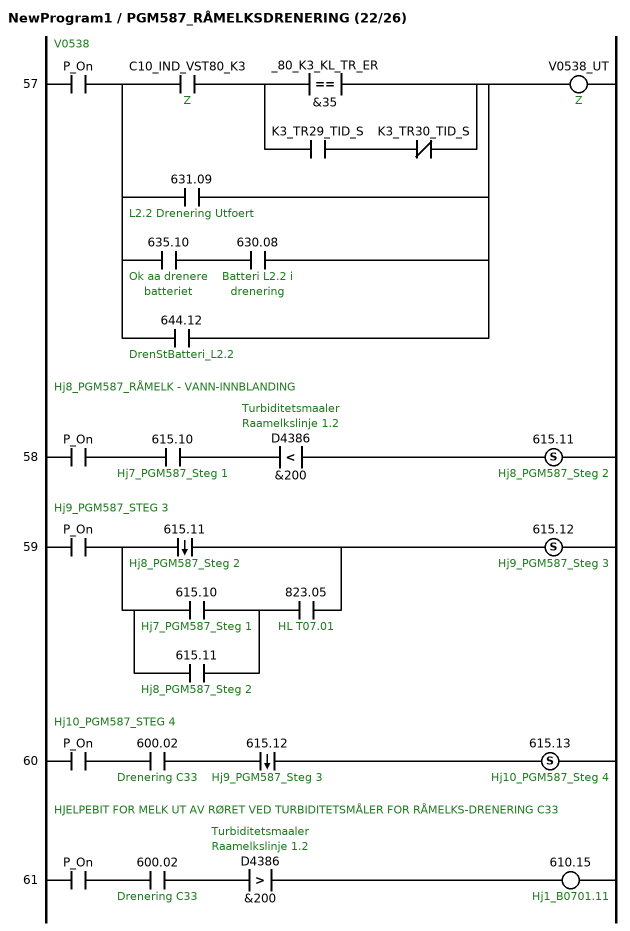
; [picture p744: NewProgram1 / PGM587_RÅMELKSDRENERING, rungs 57-61]
; rung 57: V0538
LD P_On
LD C10_IND_VST80_K3  ; Z
LD=(300) _80_K3_KL_TR_ER &35
LD K3_TR29_TID_S
ANDNOT K3_TR30_TID_S
ORLD
ANDLD
OR 631.09  ; L2.2 Drenering Utfoert
LD 635.10  ; Ok aa drenere batteriet
AND 630.08  ; Batteri L2.2 i drenering
ORLD
OR 644.12  ; DrenStBatteri_L2.2
ANDLD
OUT V0538_UT  ; Z
; rung 58: Hj8_PGM587_RÅMELK - VANN-INNBLANDING
LD P_On
AND 615.10  ; Hj7_PGM587_Steg 1
AND<(310) D4386 &200  ; Turbiditetsmaaler Raamelkslinje 1.2
SET 615.11  ; Hj8_PGM587_Steg 2
; rung 59: Hj9_PGM587_STEG 3
LD P_On
%LD 615.11  ; Hj8_PGM587_Steg 2
LD 615.10  ; Hj7_PGM587_Steg 1
OR 615.11  ; Hj8_PGM587_Steg 2
AND 823.05  ; HL T07.01
ORLD
ANDLD
SET 615.12  ; Hj9_PGM587_Steg 3
; rung 60: Hj10_PGM587_STEG 4
LD P_On
AND 600.02  ; Drenering C33
%AND 615.12  ; Hj9_PGM587_Steg 3
SET 615.13  ; Hj10_PGM587_Steg 4
; rung 61: HJELPEBIT FOR MELK UT AV RØRET VED TURBIDITETSMÅLER FOR RÅMELKS-DRENERING C33
LD P_On
AND 600.02  ; Drenering C33
AND>(320) D4386 &200  ; Turbiditetsmaaler Raamelkslinje 1.2
OUT 610.15  ; Hj1_B0701.11

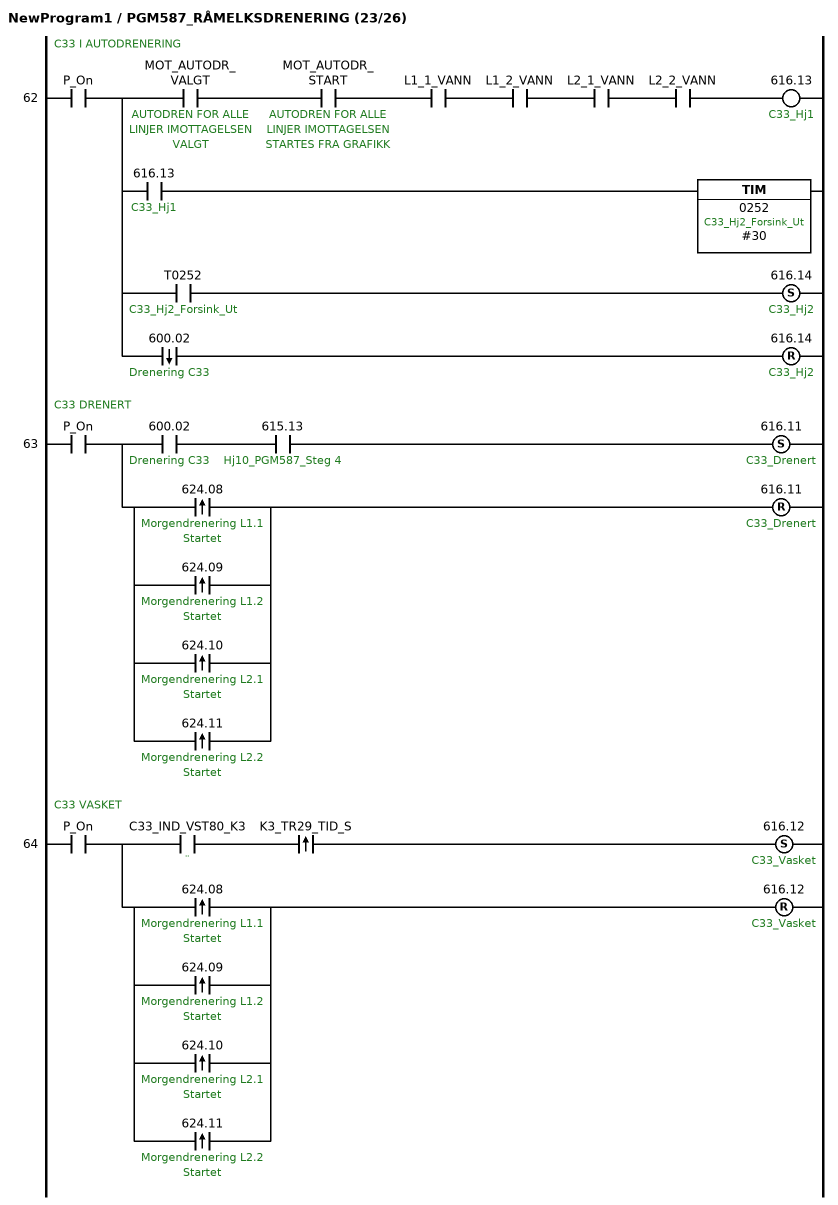
; rung 62: C33 I AUTODRENERING
LD P_On
OUT TR0
AND MOT_AUTODR_VALGT  ; AUTODREN FOR ALLE LINJER IMOTTAGELSEN VALGT
AND MOT_AUTODR_START  ; AUTODREN FOR ALLE LINJER IMOTTAGELSEN STARTES FRA GRAFIKK
AND L1_1_VANN
AND L1_2_VANN
AND L2_1_VANN
AND L2_2_VANN
OUT 616.13  ; C33_Hj1
LD TR0
AND 616.13  ; C33_Hj1
TIM 0252 #30  ; C33_Hj2_Forsink_Ut
LD TR0
AND T0252  ; C33_Hj2_Forsink_Ut
SET 616.14  ; C33_Hj2
LD TR0
%AND 600.02  ; Drenering C33
RSET 616.14  ; C33_Hj2
; rung 63: C33 DRENERT
LD P_On
OUT TR0
AND 600.02  ; Drenering C33
AND 615.13  ; Hj10_PGM587_Steg 4
SET 616.11  ; C33_Drenert
LD TR0
@LD 624.08  ; Morgendrenering L1.1 Startet
@OR 624.09  ; Morgendrenering L1.2 Startet
@OR 624.10  ; Morgendrenering L2.1 Startet
@OR 624.11  ; Morgendrenering L2.2 Startet
ANDLD
RSET 616.11  ; C33_Drenert
; rung 64: C33 VASKET
LD P_On
OUT TR0
AND C33_IND_VST80_K3  ; ¨
@AND K3_TR29_TID_S
SET 616.12  ; C33_Vasket
LD TR0
@LD 624.08  ; Morgendrenering L1.1 Startet
@OR 624.09  ; Morgendrenering L1.2 Startet
@OR 624.10  ; Morgendrenering L2.1 Startet
@OR 624.11  ; Morgendrenering L2.2 Startet
ANDLD
RSET 616.12  ; C33_Vasket

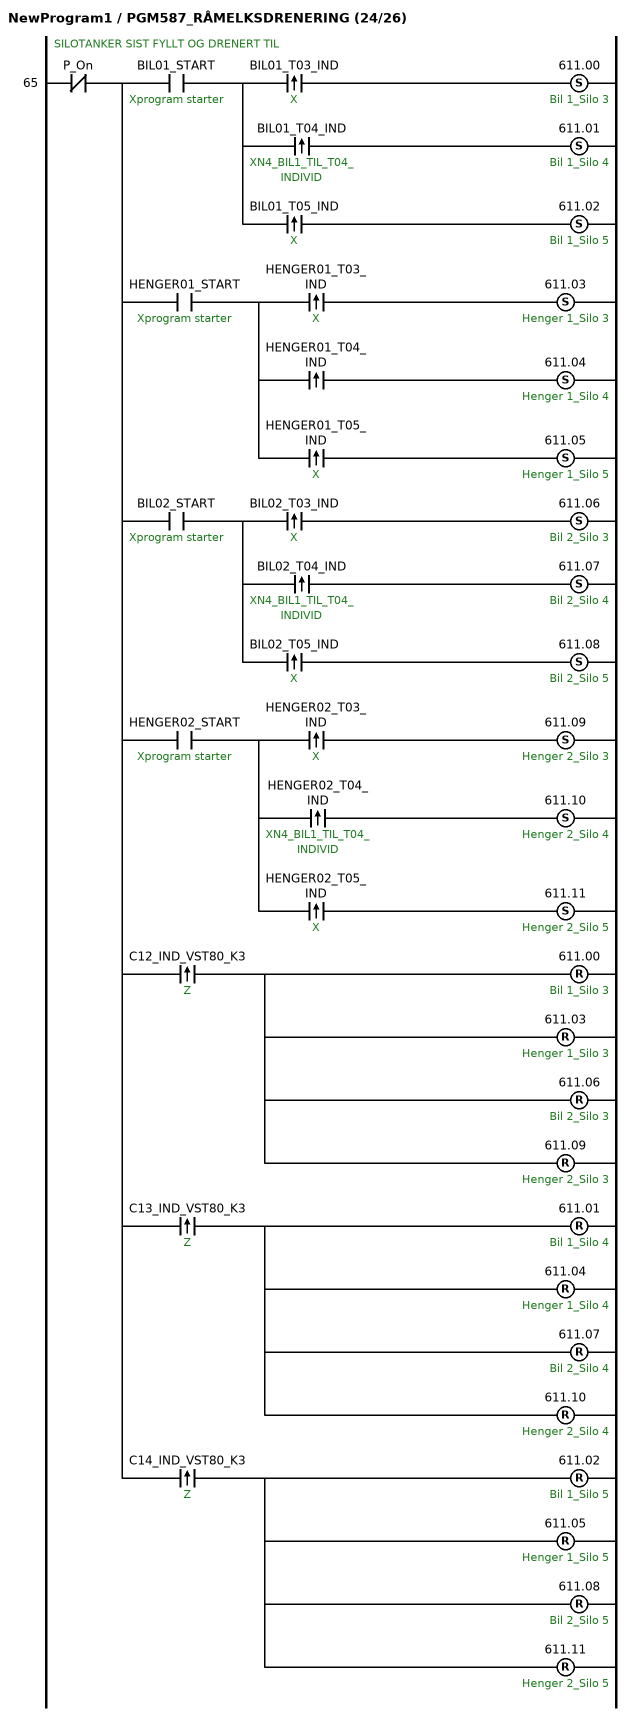
; rung 65: SILOTANKER SIST FYLLT OG DRENERT TIL
LDNOT P_On
OUT TR0
AND BIL01_START  ; Xprogram starter
OUT TR1
@AND BIL01_T03_IND  ; X
SET 611.00  ; Bil 1_Silo 3
LD TR1
@AND BIL01_T04_IND  ; XN4_BIL1_TIL_T04_INDIVID
SET 611.01  ; Bil 1_Silo 4
LD TR1
@AND BIL01_T05_IND  ; X
SET 611.02  ; Bil 1_Silo 5
LD TR0
AND HENGER01_START  ; Xprogram starter
OUT TR1
@AND HENGER01_T03_IND  ; X
SET 611.03  ; Henger 1_Silo 3
LD TR1
@AND HENGER01_T04_IND
SET 611.04  ; Henger 1_Silo 4
LD TR1
@AND HENGER01_T05_IND  ; X
SET 611.05  ; Henger 1_Silo 5
LD TR0
AND BIL02_START  ; Xprogram starter
OUT TR1
@AND BIL02_T03_IND  ; X
SET 611.06  ; Bil 2_Silo 3
LD TR1
@AND BIL02_T04_IND  ; XN4_BIL1_TIL_T04_INDIVID
SET 611.07  ; Bil 2_Silo 4
LD TR1
@AND BIL02_T05_IND  ; X
SET 611.08  ; Bil 2_Silo 5
LD TR0
AND HENGER02_START  ; Xprogram starter
OUT TR1
@AND HENGER02_T03_IND  ; X
SET 611.09  ; Henger 2_Silo 3
LD TR1
@AND HENGER02_T04_IND  ; XN4_BIL1_TIL_T04_INDIVID
SET 611.10  ; Henger 2_Silo 4
LD TR1
@AND HENGER02_T05_IND  ; X
SET 611.11  ; Henger 2_Silo 5
LD TR0
@AND C12_IND_VST80_K3  ; Z
RSET 611.00  ; Bil 1_Silo 3
RSET 611.03  ; Henger 1_Silo 3
RSET 611.06  ; Bil 2_Silo 3
RSET 611.09  ; Henger 2_Silo 3
LD TR0
@AND C13_IND_VST80_K3  ; Z
RSET 611.01  ; Bil 1_Silo 4
RSET 611.04  ; Henger 1_Silo 4
RSET 611.07  ; Bil 2_Silo 4
RSET 611.10  ; Henger 2_Silo 4
LD TR0
@AND C14_IND_VST80_K3  ; Z
RSET 611.02  ; Bil 1_Silo 5
RSET 611.05  ; Henger 1_Silo 5
RSET 611.08  ; Bil 2_Silo 5
RSET 611.11  ; Henger 2_Silo 5

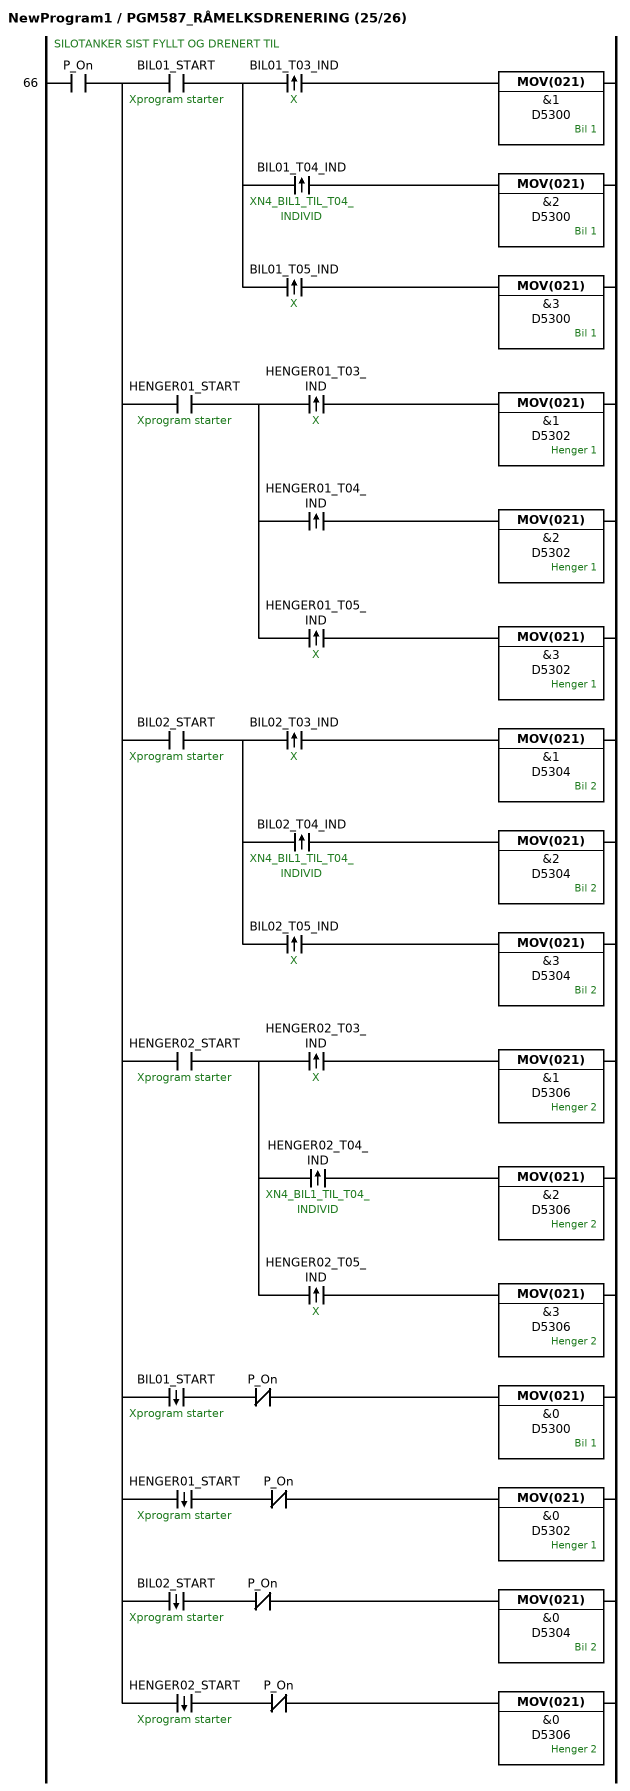
; rung 66: SILOTANKER SIST FYLLT OG DRENERT TIL
LD P_On
OUT TR0
AND BIL01_START  ; Xprogram starter
OUT TR1
@AND BIL01_T03_IND  ; X
MOV(021) &1 D5300  ; Bil 1
LD TR1
@AND BIL01_T04_IND  ; XN4_BIL1_TIL_T04_INDIVID
MOV(021) &2 D5300  ; Bil 1
LD TR1
@AND BIL01_T05_IND  ; X
MOV(021) &3 D5300  ; Bil 1
LD TR0
AND HENGER01_START  ; Xprogram starter
OUT TR1
@AND HENGER01_T03_IND  ; X
MOV(021) &1 D5302  ; Henger 1
LD TR1
@AND HENGER01_T04_IND
MOV(021) &2 D5302  ; Henger 1
LD TR1
@AND HENGER01_T05_IND  ; X
MOV(021) &3 D5302  ; Henger 1
LD TR0
AND BIL02_START  ; Xprogram starter
OUT TR1
@AND BIL02_T03_IND  ; X
MOV(021) &1 D5304  ; Bil 2
LD TR1
@AND BIL02_T04_IND  ; XN4_BIL1_TIL_T04_INDIVID
MOV(021) &2 D5304  ; Bil 2
LD TR1
@AND BIL02_T05_IND  ; X
MOV(021) &3 D5304  ; Bil 2
LD TR0
AND HENGER02_START  ; Xprogram starter
OUT TR1
@AND HENGER02_T03_IND  ; X
MOV(021) &1 D5306  ; Henger 2
LD TR1
@AND HENGER02_T04_IND  ; XN4_BIL1_TIL_T04_INDIVID
MOV(021) &2 D5306  ; Henger 2
LD TR1
@AND HENGER02_T05_IND  ; X
MOV(021) &3 D5306  ; Henger 2
LD TR0
%AND BIL01_START  ; Xprogram starter
ANDNOT P_On
MOV(021) &0 D5300  ; Bil 1
LD TR0
%AND HENGER01_START  ; Xprogram starter
ANDNOT P_On
MOV(021) &0 D5302  ; Henger 1
LD TR0
%AND BIL02_START  ; Xprogram starter
ANDNOT P_On
MOV(021) &0 D5304  ; Bil 2
LD TR0
%AND HENGER02_START  ; Xprogram starter
ANDNOT P_On
MOV(021) &0 D5306  ; Henger 2

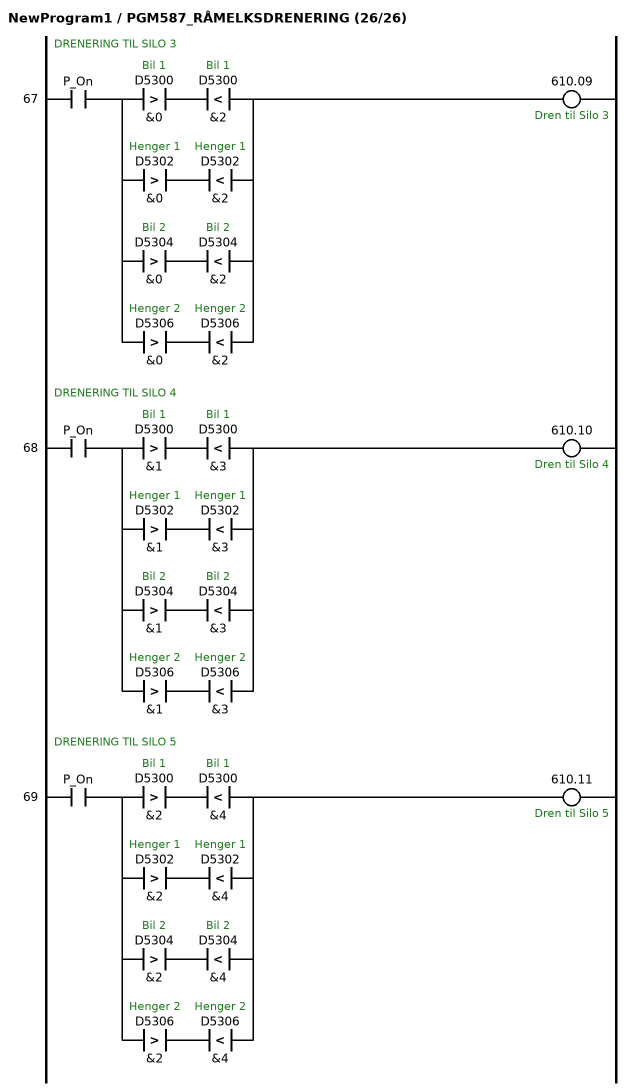
; rung 67: DRENERING TIL SILO 3
LD P_On
LD>(320) D5300 &0  ; Bil 1
AND<(310) D5300 &2  ; Bil 1
LD>(320) D5302 &0  ; Henger 1
AND<(310) D5302 &2  ; Henger 1
ORLD
LD>(320) D5304 &0  ; Bil 2
AND<(310) D5304 &2  ; Bil 2
ORLD
LD>(320) D5306 &0  ; Henger 2
AND<(310) D5306 &2  ; Henger 2
ORLD
ANDLD
OUT 610.09  ; Dren til Silo 3
; rung 68: DRENERING TIL SILO 4
LD P_On
LD>(320) D5300 &1  ; Bil 1
AND<(310) D5300 &3  ; Bil 1
LD>(320) D5302 &1  ; Henger 1
AND<(310) D5302 &3  ; Henger 1
ORLD
LD>(320) D5304 &1  ; Bil 2
AND<(310) D5304 &3  ; Bil 2
ORLD
LD>(320) D5306 &1  ; Henger 2
AND<(310) D5306 &3  ; Henger 2
ORLD
ANDLD
OUT 610.10  ; Dren til Silo 4
; rung 69: DRENERING TIL SILO 5
LD P_On
LD>(320) D5300 &2  ; Bil 1
AND<(310) D5300 &4  ; Bil 1
LD>(320) D5302 &2  ; Henger 1
AND<(310) D5302 &4  ; Henger 1
ORLD
LD>(320) D5304 &2  ; Bil 2
AND<(310) D5304 &4  ; Bil 2
ORLD
LD>(320) D5306 &2  ; Henger 2
AND<(310) D5306 &4  ; Henger 2
ORLD
ANDLD
OUT 610.11  ; Dren til Silo 5

### Section PGM588_DEPONI_T27_03

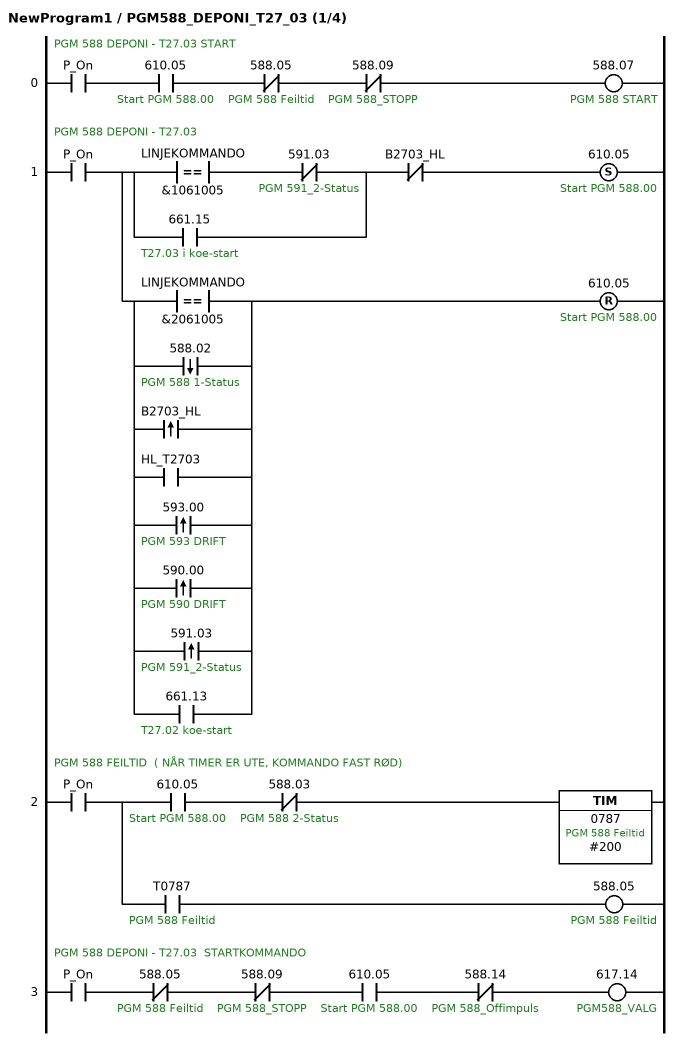
; rung 0: PGM 588 DEPONI - T27.03 START
LD P_On
AND 610.05  ; Start PGM 588.00
ANDNOT 588.05  ; PGM 588 Feiltid
ANDNOT 588.09  ; PGM 588_STOPP
OUT 588.07  ; PGM 588 START
; rung 1: PGM 588 DEPONI - T27.03
LD P_On
OUT TR0
LD=L(301) LINJEKOMMANDO &1061005
ANDNOT 591.03  ; PGM 591_2-Status
OR 661.15  ; T27.03 i koe-start
ANDLD
ANDNOT B2703_HL
SET 610.05  ; Start PGM 588.00
LD TR0
LD=L(301) LINJEKOMMANDO &2061005
%OR 588.02  ; PGM 588 1-Status
@OR B2703_HL
OR HL_T2703
@OR 593.00  ; PGM 593 DRIFT
@OR 590.00  ; PGM 590 DRIFT
@OR 591.03  ; PGM 591_2-Status
OR 661.13  ; T27.02 koe-start
ANDLD
RSET 610.05  ; Start PGM 588.00
; rung 2: PGM 588 FEILTID  ( NÅR TIMER ER UTE, KOMMANDO FAST RØD)
LD P_On
OUT TR0
AND 610.05  ; Start PGM 588.00
ANDNOT 588.03  ; PGM 588 2-Status
TIM 0787 #200  ; PGM 588 Feiltid
LD TR0
AND T0787  ; PGM 588 Feiltid
OUT 588.05  ; PGM 588 Feiltid
; rung 3: PGM 588 DEPONI - T27.03  STARTKOMMANDO
LD P_On
ANDNOT 588.05  ; PGM 588 Feiltid
ANDNOT 588.09  ; PGM 588_STOPP
AND 610.05  ; Start PGM 588.00
ANDNOT 588.14  ; PGM 588_Offimpuls
OUT 617.14  ; PGM588_VALG

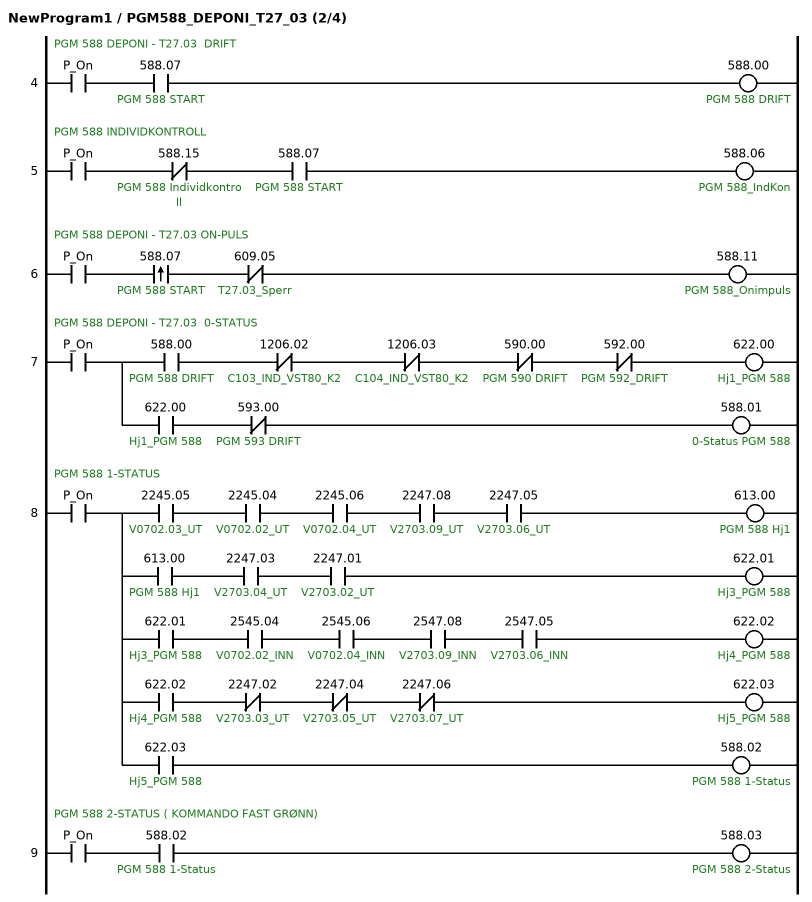
; rung 4: PGM 588 DEPONI - T27.03  DRIFT
LD P_On
AND 588.07  ; PGM 588 START
OUT 588.00  ; PGM 588 DRIFT
; rung 5: PGM 588 INDIVIDKONTROLL
LD P_On
ANDNOT 588.15  ; PGM 588 Individkontroll
AND 588.07  ; PGM 588 START
OUT 588.06  ; PGM 588_IndKon
; rung 6: PGM 588 DEPONI - T27.03 ON-PULS
LD P_On
@AND 588.07  ; PGM 588 START
ANDNOT 609.05  ; T27.03_Sperr
OUT 588.11  ; PGM 588_Onimpuls
; rung 7: PGM 588 DEPONI - T27.03  0-STATUS
LD P_On
OUT TR0
AND 588.00  ; PGM 588 DRIFT
ANDNOT 1206.02  ; C103_IND_VST80_K2
ANDNOT 1206.03  ; C104_IND_VST80_K2
ANDNOT 590.00  ; PGM 590 DRIFT
ANDNOT 592.00  ; PGM 592_DRIFT
OUT 622.00  ; Hj1_PGM 588
LD TR0
AND 622.00  ; Hj1_PGM 588
ANDNOT 593.00  ; PGM 593 DRIFT
OUT 588.01  ; 0-Status PGM 588
; rung 8: PGM 588 1-STATUS
LD P_On
OUT TR0
AND 2245.05  ; V0702.03_UT
AND 2245.04  ; V0702.02_UT
AND 2245.06  ; V0702.04_UT
AND 2247.08  ; V2703.09_UT
AND 2247.05  ; V2703.06_UT
OUT 613.00  ; PGM 588 Hj1
LD TR0
AND 613.00  ; PGM 588 Hj1
AND 2247.03  ; V2703.04_UT
AND 2247.01  ; V2703.02_UT
OUT 622.01  ; Hj3_PGM 588
LD TR0
AND 622.01  ; Hj3_PGM 588
AND 2545.04  ; V0702.02_INN
AND 2545.06  ; V0702.04_INN
AND 2547.08  ; V2703.09_INN
AND 2547.05  ; V2703.06_INN
OUT 622.02  ; Hj4_PGM 588
LD TR0
AND 622.02  ; Hj4_PGM 588
ANDNOT 2247.02  ; V2703.03_UT
ANDNOT 2247.04  ; V2703.05_UT
ANDNOT 2247.06  ; V2703.07_UT
OUT 622.03  ; Hj5_PGM 588
LD TR0
AND 622.03  ; Hj5_PGM 588
OUT 588.02  ; PGM 588 1-Status
; rung 9: PGM 588 2-STATUS ( KOMMANDO FAST GRØNN)
LD P_On
AND 588.02  ; PGM 588 1-Status
OUT 588.03  ; PGM 588 2-Status

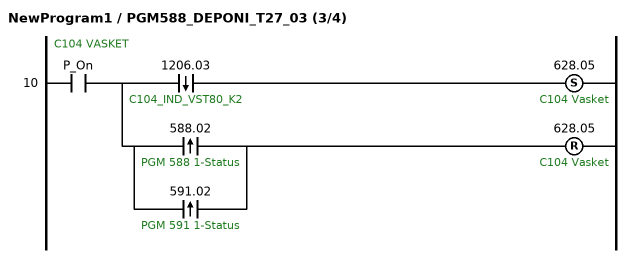
; rung 10: C104 VASKET
LD P_On
OUT TR0
%AND 1206.03  ; C104_IND_VST80_K2
SET 628.05  ; C104 Vasket
LD TR0
@LD 588.02  ; PGM 588 1-Status
@OR 591.02  ; PGM 591 1-Status
ANDLD
RSET 628.05  ; C104 Vasket

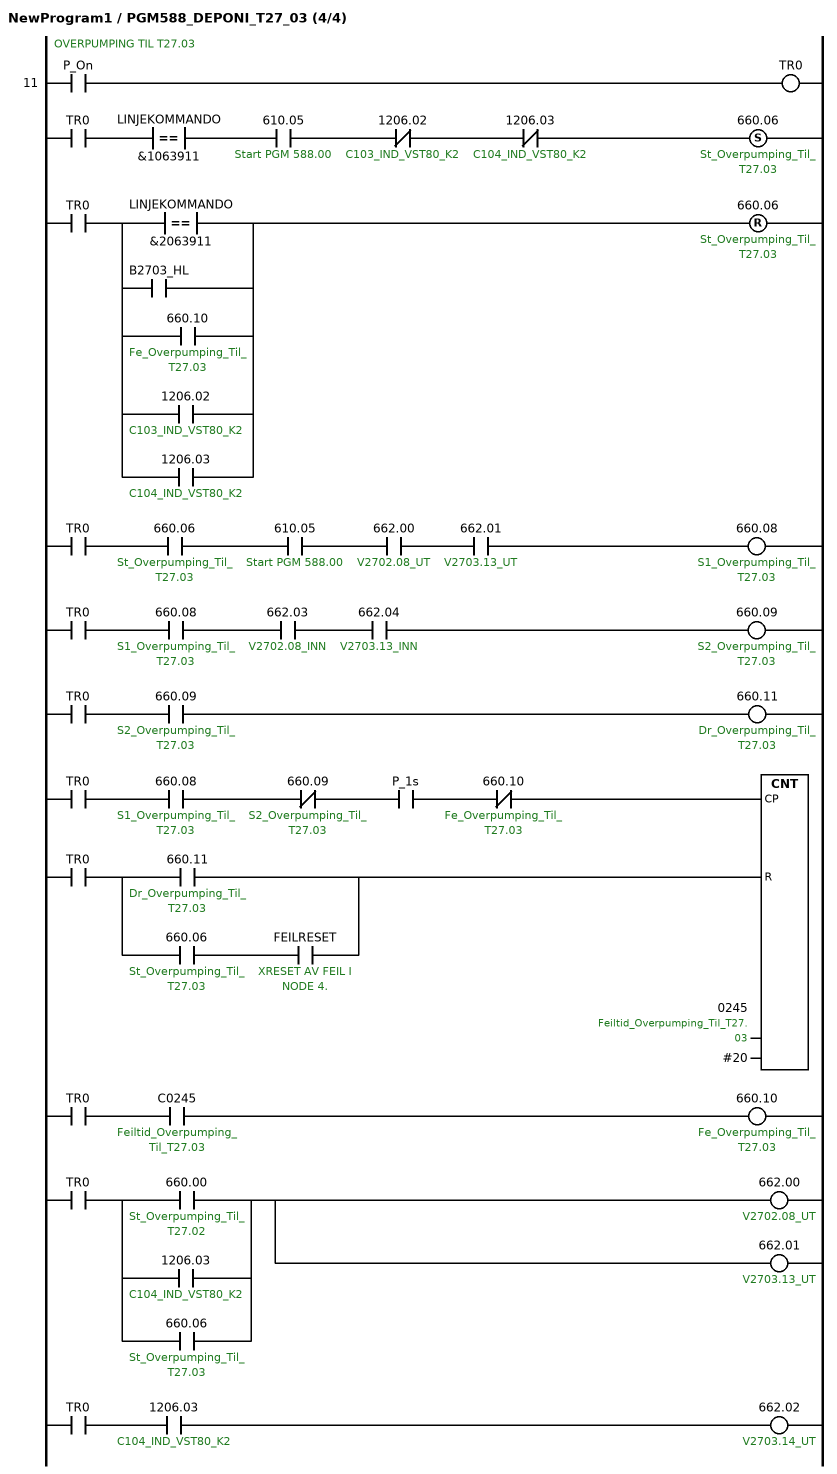
; rung 11: OVERPUMPING TIL T27.03
LD P_On
OUT TR0
AND=L(301) LINJEKOMMANDO &1063911
AND 610.05  ; Start PGM 588.00
ANDNOT 1206.02  ; C103_IND_VST80_K2
ANDNOT 1206.03  ; C104_IND_VST80_K2
SET 660.06  ; St_Overpumping_Til_T27.03
LD TR0
LD=L(301) LINJEKOMMANDO &2063911
OR B2703_HL
OR 660.10  ; Fe_Overpumping_Til_T27.03
OR 1206.02  ; C103_IND_VST80_K2
OR 1206.03  ; C104_IND_VST80_K2
ANDLD
RSET 660.06  ; St_Overpumping_Til_T27.03
LD TR0
AND 660.06  ; St_Overpumping_Til_T27.03
AND 610.05  ; Start PGM 588.00
AND 662.00  ; V2702.08_UT
AND 662.01  ; V2703.13_UT
OUT 660.08  ; S1_Overpumping_Til_T27.03
LD TR0
AND 660.08  ; S1_Overpumping_Til_T27.03
AND 662.03  ; V2702.08_INN
AND 662.04  ; V2703.13_INN
OUT 660.09  ; S2_Overpumping_Til_T27.03
LD TR0
AND 660.09  ; S2_Overpumping_Til_T27.03
OUT 660.11  ; Dr_Overpumping_Til_T27.03
LD TR0
AND 660.08  ; S1_Overpumping_Til_T27.03
ANDNOT 660.09  ; S2_Overpumping_Til_T27.03
AND P_1s
ANDNOT 660.10  ; Fe_Overpumping_Til_T27.03
LD TR0
LD 660.11  ; Dr_Overpumping_Til_T27.03
LD 660.06  ; St_Overpumping_Til_T27.03
AND FEILRESET  ; XRESET AV FEIL I NODE 4.
ORLD
ANDLD
CNT 0245 #20  ; Feiltid_Overpumping_Til_T27.03
LD TR0
AND C0245  ; Feiltid_Overpumping_Til_T27.03
OUT 660.10  ; Fe_Overpumping_Til_T27.03
LD TR0
LD 660.00  ; St_Overpumping_Til_T27.02
OR 1206.03  ; C104_IND_VST80_K2
OR 660.06  ; St_Overpumping_Til_T27.03
ANDLD
OUT 662.00  ; V2702.08_UT
OUT 662.01  ; V2703.13_UT
LD TR0
AND 1206.03  ; C104_IND_VST80_K2
OUT 662.02  ; V2703.14_UT

### Section PGM589_T27_02

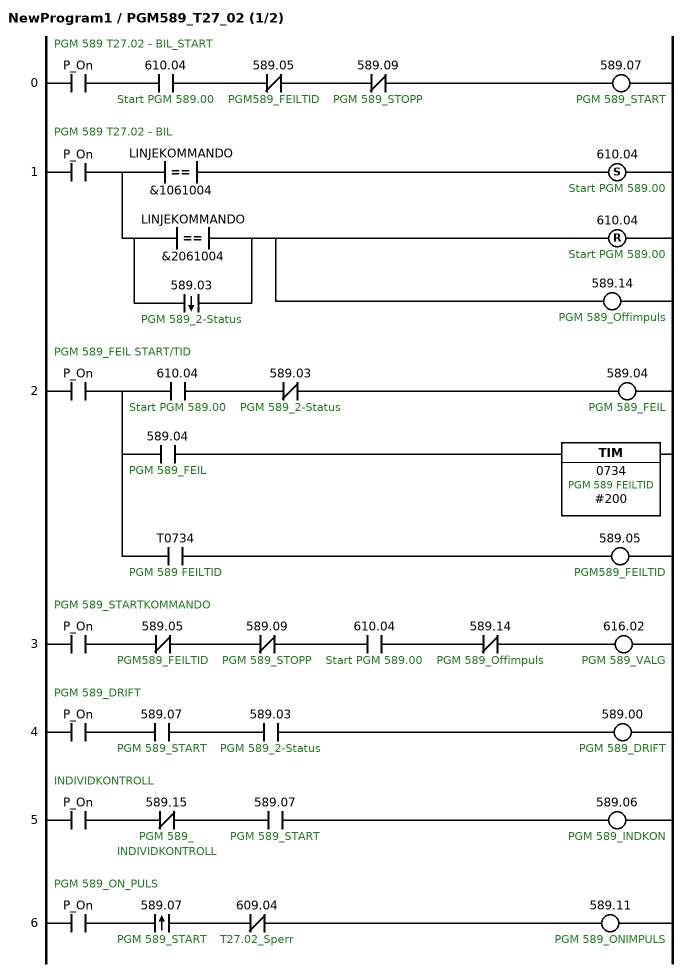
; rung 0: PGM 589 T27.02 - BIL_START
LD P_On
AND 610.04  ; Start PGM 589.00
ANDNOT 589.05  ; PGM589_FEILTID
ANDNOT 589.09  ; PGM 589_STOPP
OUT 589.07  ; PGM 589_START
; rung 1: PGM 589 T27.02 - BIL
LD P_On
OUT TR0
AND=L(301) LINJEKOMMANDO &1061004
SET 610.04  ; Start PGM 589.00
LD TR0
LD=L(301) LINJEKOMMANDO &2061004
%OR 589.03  ; PGM 589_2-Status
ANDLD
RSET 610.04  ; Start PGM 589.00
OUT 589.14  ; PGM 589_Offimpuls
; rung 2: PGM 589_FEIL START/TID
LD P_On
OUT TR0
AND 610.04  ; Start PGM 589.00
ANDNOT 589.03  ; PGM 589_2-Status
OUT 589.04  ; PGM 589_FEIL
LD TR0
AND 589.04  ; PGM 589_FEIL
TIM 0734 #200  ; PGM 589 FEILTID
LD TR0
AND T0734  ; PGM 589 FEILTID
OUT 589.05  ; PGM589_FEILTID
; rung 3: PGM 589_STARTKOMMANDO
LD P_On
ANDNOT 589.05  ; PGM589_FEILTID
ANDNOT 589.09  ; PGM 589_STOPP
AND 610.04  ; Start PGM 589.00
ANDNOT 589.14  ; PGM 589_Offimpuls
OUT 616.02  ; PGM 589_VALG
; rung 4: PGM 589_DRIFT
LD P_On
AND 589.07  ; PGM 589_START
AND 589.03  ; PGM 589_2-Status
OUT 589.00  ; PGM 589_DRIFT
; rung 5: INDIVIDKONTROLL
LD P_On
ANDNOT 589.15  ; PGM 589_INDIVIDKONTROLL
AND 589.07  ; PGM 589_START
OUT 589.06  ; PGM 589_INDKON
; rung 6: PGM 589_ON_PULS
LD P_On
@AND 589.07  ; PGM 589_START
ANDNOT 609.04  ; T27.02_Sperr
OUT 589.11  ; PGM 589_ONIMPULS

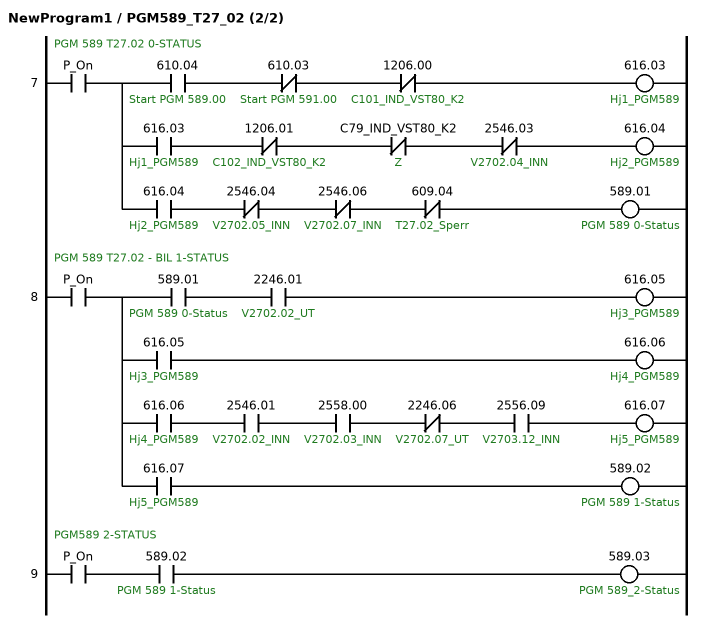
; rung 7: PGM 589 T27.02 0-STATUS
LD P_On
OUT TR0
AND 610.04  ; Start PGM 589.00
ANDNOT 610.03  ; Start PGM 591.00
ANDNOT 1206.00  ; C101_IND_VST80_K2
OUT 616.03  ; Hj1_PGM589
LD TR0
AND 616.03  ; Hj1_PGM589
ANDNOT 1206.01  ; C102_IND_VST80_K2
ANDNOT C79_IND_VST80_K2  ; Z
ANDNOT 2546.03  ; V2702.04_INN
OUT 616.04  ; Hj2_PGM589
LD TR0
AND 616.04  ; Hj2_PGM589
ANDNOT 2546.04  ; V2702.05_INN
ANDNOT 2546.06  ; V2702.07_INN
ANDNOT 609.04  ; T27.02_Sperr
OUT 589.01  ; PGM 589 0-Status
; rung 8: PGM 589 T27.02 - BIL 1-STATUS
LD P_On
OUT TR0
AND 589.01  ; PGM 589 0-Status
AND 2246.01  ; V2702.02_UT
OUT 616.05  ; Hj3_PGM589
LD TR0
AND 616.05  ; Hj3_PGM589
OUT 616.06  ; Hj4_PGM589
LD TR0
AND 616.06  ; Hj4_PGM589
AND 2546.01  ; V2702.02_INN
AND 2558.00  ; V2702.03_INN
ANDNOT 2246.06  ; V2702.07_UT
AND 2556.09  ; V2703.12_INN
OUT 616.07  ; Hj5_PGM589
LD TR0
AND 616.07  ; Hj5_PGM589
OUT 589.02  ; PGM 589 1-Status
; rung 9: PGM589 2-STATUS
LD P_On
AND 589.02  ; PGM 589 1-Status
OUT 589.03  ; PGM 589_2-Status

### Section PGM590_T27_03_BIL

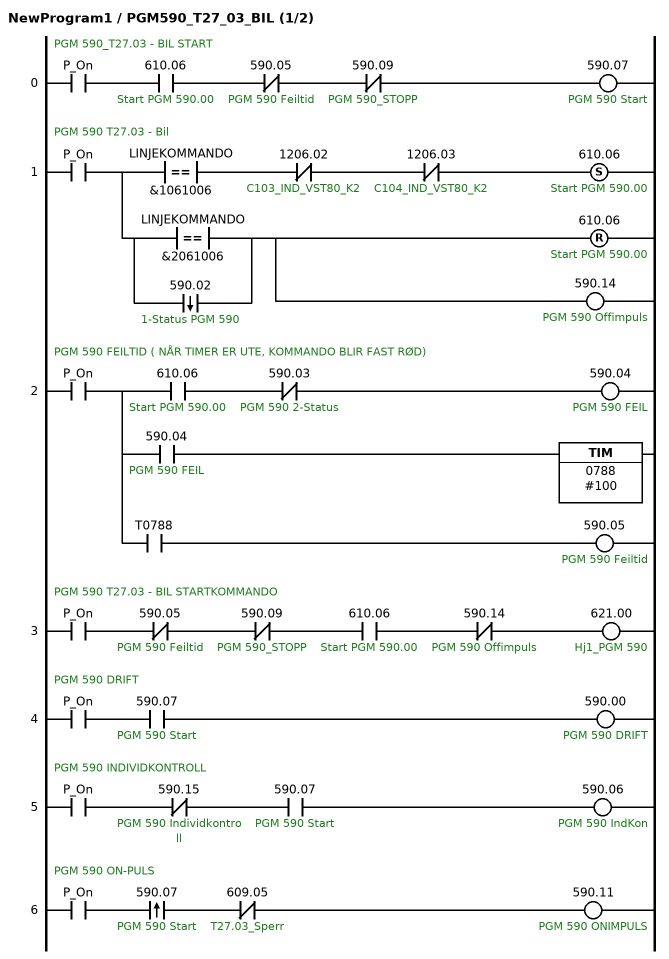
; rung 0: PGM 590_T27.03 - BIL START
LD P_On
AND 610.06  ; Start PGM 590.00
ANDNOT 590.05  ; PGM 590 Feiltid
ANDNOT 590.09  ; PGM 590_STOPP
OUT 590.07  ; PGM 590 Start
; rung 1: PGM 590 T27.03 - Bil
LD P_On
OUT TR0
AND=L(301) LINJEKOMMANDO &1061006
ANDNOT 1206.02  ; C103_IND_VST80_K2
ANDNOT 1206.03  ; C104_IND_VST80_K2
SET 610.06  ; Start PGM 590.00
LD TR0
LD=L(301) LINJEKOMMANDO &2061006
%OR 590.02  ; 1-Status PGM 590
ANDLD
RSET 610.06  ; Start PGM 590.00
OUT 590.14  ; PGM 590 Offimpuls
; rung 2: PGM 590 FEILTID ( NÅR TIMER ER UTE, KOMMANDO BLIR FAST RØD)
LD P_On
OUT TR0
AND 610.06  ; Start PGM 590.00
ANDNOT 590.03  ; PGM 590 2-Status
OUT 590.04  ; PGM 590 FEIL
LD TR0
AND 590.04  ; PGM 590 FEIL
TIM 0788 #100
LD TR0
AND T0788
OUT 590.05  ; PGM 590 Feiltid
; rung 3: PGM 590 T27.03 - BIL STARTKOMMANDO
LD P_On
ANDNOT 590.05  ; PGM 590 Feiltid
ANDNOT 590.09  ; PGM 590_STOPP
AND 610.06  ; Start PGM 590.00
ANDNOT 590.14  ; PGM 590 Offimpuls
OUT 621.00  ; Hj1_PGM 590
; rung 4: PGM 590 DRIFT
LD P_On
AND 590.07  ; PGM 590 Start
OUT 590.00  ; PGM 590 DRIFT
; rung 5: PGM 590 INDIVIDKONTROLL
LD P_On
ANDNOT 590.15  ; PGM 590 Individkontroll
AND 590.07  ; PGM 590 Start
OUT 590.06  ; PGM 590 IndKon
; rung 6: PGM 590 ON-PULS
LD P_On
@AND 590.07  ; PGM 590 Start
ANDNOT 609.05  ; T27.03_Sperr
OUT 590.11  ; PGM 590 ONIMPULS

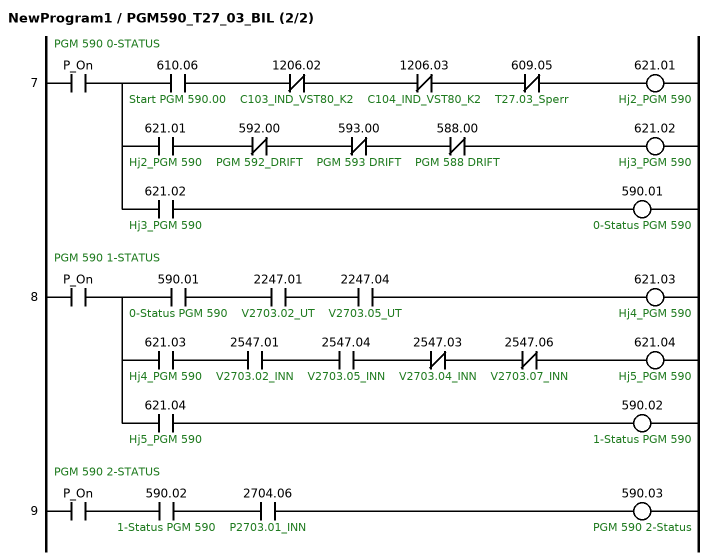
; rung 7: PGM 590 0-STATUS
LD P_On
OUT TR0
AND 610.06  ; Start PGM 590.00
ANDNOT 1206.02  ; C103_IND_VST80_K2
ANDNOT 1206.03  ; C104_IND_VST80_K2
ANDNOT 609.05  ; T27.03_Sperr
OUT 621.01  ; Hj2_PGM 590
LD TR0
AND 621.01  ; Hj2_PGM 590
ANDNOT 592.00  ; PGM 592_DRIFT
ANDNOT 593.00  ; PGM 593 DRIFT
ANDNOT 588.00  ; PGM 588 DRIFT
OUT 621.02  ; Hj3_PGM 590
LD TR0
AND 621.02  ; Hj3_PGM 590
OUT 590.01  ; 0-Status PGM 590
; rung 8: PGM 590 1-STATUS
LD P_On
OUT TR0
AND 590.01  ; 0-Status PGM 590
AND 2247.01  ; V2703.02_UT
AND 2247.04  ; V2703.05_UT
OUT 621.03  ; Hj4_PGM 590
LD TR0
AND 621.03  ; Hj4_PGM 590
AND 2547.01  ; V2703.02_INN
AND 2547.04  ; V2703.05_INN
ANDNOT 2547.03  ; V2703.04_INN
ANDNOT 2547.06  ; V2703.07_INN
OUT 621.04  ; Hj5_PGM 590
LD TR0
AND 621.04  ; Hj5_PGM 590
OUT 590.02  ; 1-Status PGM 590
; rung 9: PGM 590 2-STATUS
LD P_On
AND 590.02  ; 1-Status PGM 590
AND 2704.06  ; P2703.01_INN
OUT 590.03  ; PGM 590 2-Status

### Section PGM591_T27_02

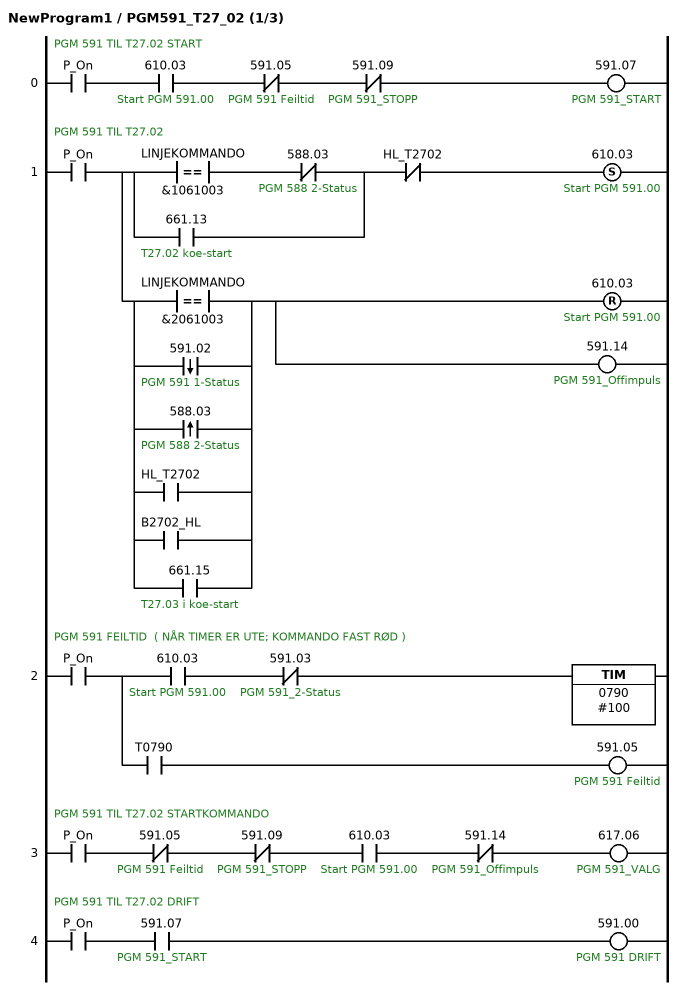
; rung 0: PGM 591 TIL T27.02 START
LD P_On
AND 610.03  ; Start PGM 591.00
ANDNOT 591.05  ; PGM 591 Feiltid
ANDNOT 591.09  ; PGM 591_STOPP
OUT 591.07  ; PGM 591_START
; rung 1: PGM 591 TIL T27.02
LD P_On
OUT TR0
LD=L(301) LINJEKOMMANDO &1061003
ANDNOT 588.03  ; PGM 588 2-Status
OR 661.13  ; T27.02 koe-start
ANDLD
ANDNOT HL_T2702
SET 610.03  ; Start PGM 591.00
LD TR0
LD=L(301) LINJEKOMMANDO &2061003
%OR 591.02  ; PGM 591 1-Status
@OR 588.03  ; PGM 588 2-Status
OR HL_T2702
OR B2702_HL
OR 661.15  ; T27.03 i koe-start
ANDLD
RSET 610.03  ; Start PGM 591.00
OUT 591.14  ; PGM 591_Offimpuls
; rung 2: PGM 591 FEILTID  ( NÅR TIMER ER UTE; KOMMANDO FAST RØD )
LD P_On
OUT TR0
AND 610.03  ; Start PGM 591.00
ANDNOT 591.03  ; PGM 591_2-Status
TIM 0790 #100
LD TR0
AND T0790
OUT 591.05  ; PGM 591 Feiltid
; rung 3: PGM 591 TIL T27.02 STARTKOMMANDO
LD P_On
ANDNOT 591.05  ; PGM 591 Feiltid
ANDNOT 591.09  ; PGM 591_STOPP
AND 610.03  ; Start PGM 591.00
ANDNOT 591.14  ; PGM 591_Offimpuls
OUT 617.06  ; PGM 591_VALG
; rung 4: PGM 591 TIL T27.02 DRIFT
LD P_On
AND 591.07  ; PGM 591_START
OUT 591.00  ; PGM 591 DRIFT

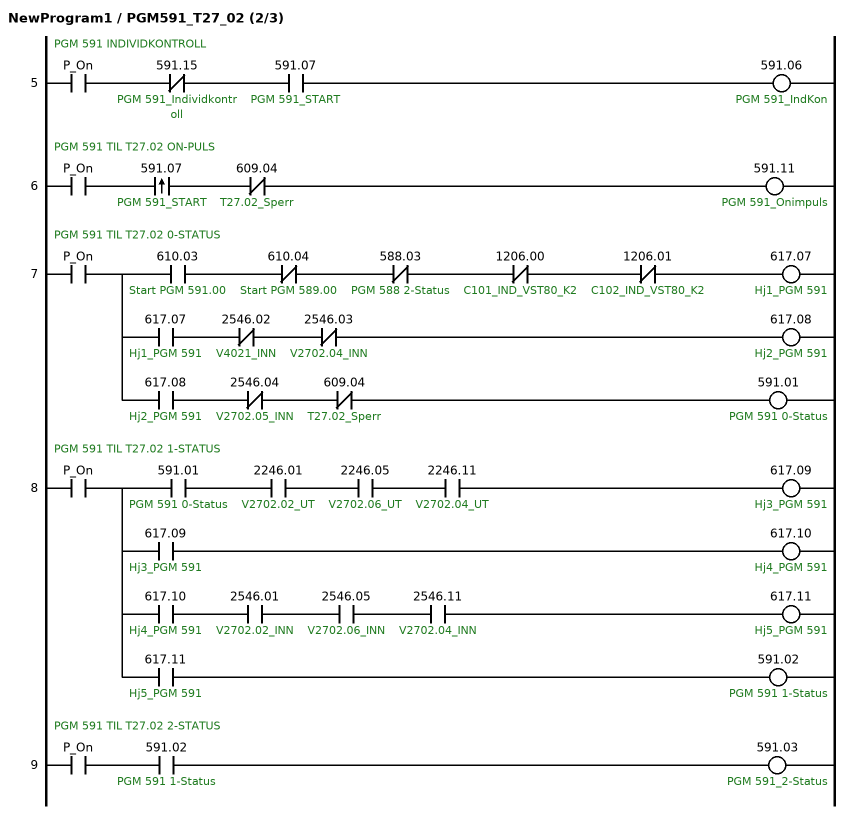
; rung 5: PGM 591 INDIVIDKONTROLL
LD P_On
ANDNOT 591.15  ; PGM 591_Individkontroll
AND 591.07  ; PGM 591_START
OUT 591.06  ; PGM 591_IndKon
; rung 6: PGM 591 TIL T27.02 ON-PULS
LD P_On
@AND 591.07  ; PGM 591_START
ANDNOT 609.04  ; T27.02_Sperr
OUT 591.11  ; PGM 591_Onimpuls
; rung 7: PGM 591 TIL T27.02 0-STATUS
LD P_On
OUT TR0
AND 610.03  ; Start PGM 591.00
ANDNOT 610.04  ; Start PGM 589.00
ANDNOT 588.03  ; PGM 588 2-Status
ANDNOT 1206.00  ; C101_IND_VST80_K2
ANDNOT 1206.01  ; C102_IND_VST80_K2
OUT 617.07  ; Hj1_PGM 591
LD TR0
AND 617.07  ; Hj1_PGM 591
ANDNOT 2546.02  ; V4021_INN
ANDNOT 2546.03  ; V2702.04_INN
OUT 617.08  ; Hj2_PGM 591
LD TR0
AND 617.08  ; Hj2_PGM 591
ANDNOT 2546.04  ; V2702.05_INN
ANDNOT 609.04  ; T27.02_Sperr
OUT 591.01  ; PGM 591 0-Status
; rung 8: PGM 591 TIL T27.02 1-STATUS
LD P_On
OUT TR0
AND 591.01  ; PGM 591 0-Status
AND 2246.01  ; V2702.02_UT
AND 2246.05  ; V2702.06_UT
AND 2246.11  ; V2702.04_UT
OUT 617.09  ; Hj3_PGM 591
LD TR0
AND 617.09  ; Hj3_PGM 591
OUT 617.10  ; Hj4_PGM 591
LD TR0
AND 617.10  ; Hj4_PGM 591
AND 2546.01  ; V2702.02_INN
AND 2546.05  ; V2702.06_INN
AND 2546.11  ; V2702.04_INN
OUT 617.11  ; Hj5_PGM 591
LD TR0
AND 617.11  ; Hj5_PGM 591
OUT 591.02  ; PGM 591 1-Status
; rung 9: PGM 591 TIL T27.02 2-STATUS
LD P_On
AND 591.02  ; PGM 591 1-Status
OUT 591.03  ; PGM 591_2-Status

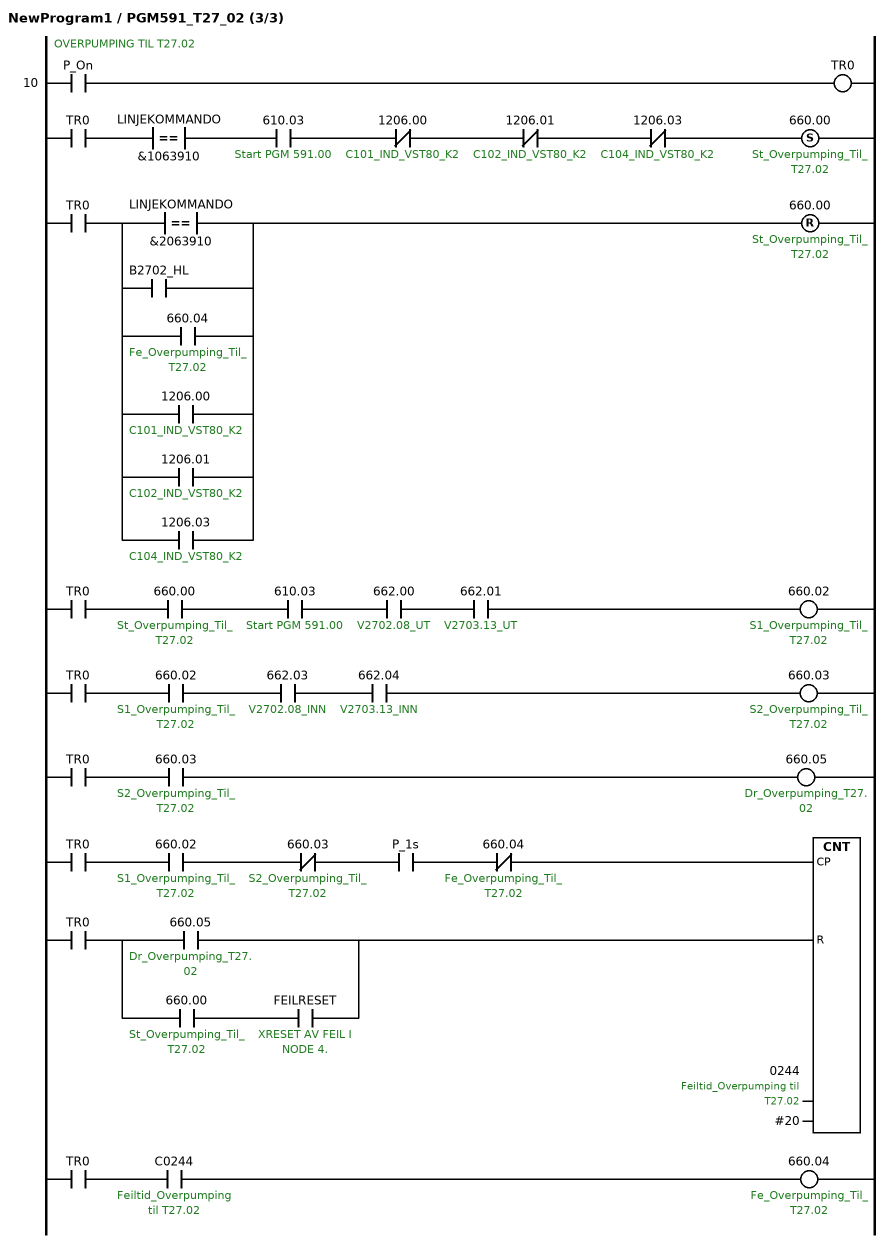
; rung 10: OVERPUMPING TIL T27.02
LD P_On
OUT TR0
AND=L(301) LINJEKOMMANDO &1063910
AND 610.03  ; Start PGM 591.00
ANDNOT 1206.00  ; C101_IND_VST80_K2
ANDNOT 1206.01  ; C102_IND_VST80_K2
ANDNOT 1206.03  ; C104_IND_VST80_K2
SET 660.00  ; St_Overpumping_Til_T27.02
LD TR0
LD=L(301) LINJEKOMMANDO &2063910
OR B2702_HL
OR 660.04  ; Fe_Overpumping_Til_T27.02
OR 1206.00  ; C101_IND_VST80_K2
OR 1206.01  ; C102_IND_VST80_K2
OR 1206.03  ; C104_IND_VST80_K2
ANDLD
RSET 660.00  ; St_Overpumping_Til_T27.02
LD TR0
AND 660.00  ; St_Overpumping_Til_T27.02
AND 610.03  ; Start PGM 591.00
AND 662.00  ; V2702.08_UT
AND 662.01  ; V2703.13_UT
OUT 660.02  ; S1_Overpumping_Til_T27.02
LD TR0
AND 660.02  ; S1_Overpumping_Til_T27.02
AND 662.03  ; V2702.08_INN
AND 662.04  ; V2703.13_INN
OUT 660.03  ; S2_Overpumping_Til_T27.02
LD TR0
AND 660.03  ; S2_Overpumping_Til_T27.02
OUT 660.05  ; Dr_Overpumping_T27.02
LD TR0
AND 660.02  ; S1_Overpumping_Til_T27.02
ANDNOT 660.03  ; S2_Overpumping_Til_T27.02
AND P_1s
ANDNOT 660.04  ; Fe_Overpumping_Til_T27.02
LD TR0
LD 660.05  ; Dr_Overpumping_T27.02
LD 660.00  ; St_Overpumping_Til_T27.02
AND FEILRESET  ; XRESET AV FEIL I NODE 4.
ORLD
ANDLD
CNT 0244 #20  ; Feiltid_Overpumping til T27.02
LD TR0
AND C0244  ; Feiltid_Overpumping til T27.02
OUT 660.04  ; Fe_Overpumping_Til_T27.02

### Section PGM592_DRENERING_T27_03

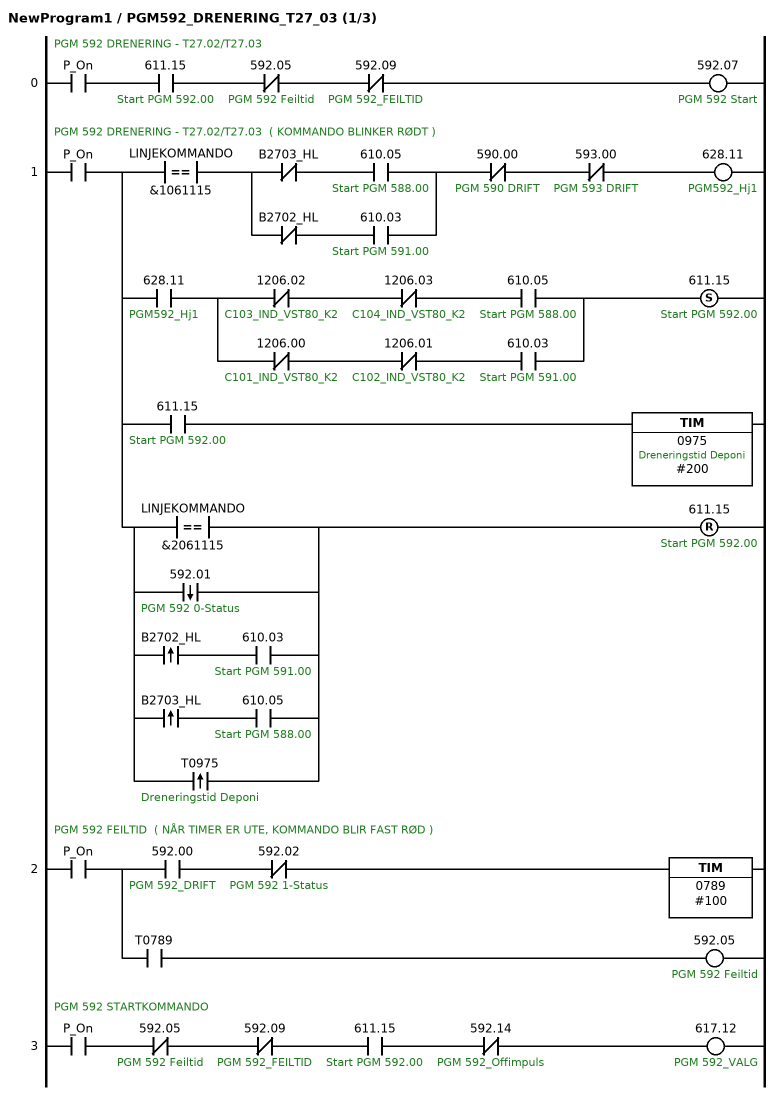
; rung 0: PGM 592 DRENERING - T27.02/T27.03
LD P_On
AND 611.15  ; Start PGM 592.00
ANDNOT 592.05  ; PGM 592 Feiltid
ANDNOT 592.09  ; PGM 592_FEILTID
OUT 592.07  ; PGM 592 Start
; rung 1: PGM 592 DRENERING - T27.02/T27.03  ( KOMMANDO BLINKER RØDT )
LD P_On
OUT TR0
AND=L(301) LINJEKOMMANDO &1061115
LDNOT B2703_HL
AND 610.05  ; Start PGM 588.00
LDNOT B2702_HL
AND 610.03  ; Start PGM 591.00
ORLD
ANDLD
ANDNOT 590.00  ; PGM 590 DRIFT
ANDNOT 593.00  ; PGM 593 DRIFT
OUT 628.11  ; PGM592_Hj1
LD TR0
AND 628.11  ; PGM592_Hj1
LDNOT 1206.02  ; C103_IND_VST80_K2
ANDNOT 1206.03  ; C104_IND_VST80_K2
AND 610.05  ; Start PGM 588.00
LDNOT 1206.00  ; C101_IND_VST80_K2
ANDNOT 1206.01  ; C102_IND_VST80_K2
AND 610.03  ; Start PGM 591.00
ORLD
ANDLD
SET 611.15  ; Start PGM 592.00
LD TR0
AND 611.15  ; Start PGM 592.00
TIM 0975 #200  ; Dreneringstid Deponi
LD TR0
LD=L(301) LINJEKOMMANDO &2061115
%OR 592.01  ; PGM 592 0-Status
@LD B2702_HL
AND 610.03  ; Start PGM 591.00
ORLD
@LD B2703_HL
AND 610.05  ; Start PGM 588.00
ORLD
@OR T0975  ; Dreneringstid Deponi
ANDLD
RSET 611.15  ; Start PGM 592.00
; rung 2: PGM 592 FEILTID  ( NÅR TIMER ER UTE, KOMMANDO BLIR FAST RØD )
LD P_On
OUT TR0
AND 592.00  ; PGM 592_DRIFT
ANDNOT 592.02  ; PGM 592 1-Status
TIM 0789 #100
LD TR0
AND T0789
OUT 592.05  ; PGM 592 Feiltid
; rung 3: PGM 592 STARTKOMMANDO
LD P_On
ANDNOT 592.05  ; PGM 592 Feiltid
ANDNOT 592.09  ; PGM 592_FEILTID
AND 611.15  ; Start PGM 592.00
ANDNOT 592.14  ; PGM 592_Offimpuls
OUT 617.12  ; PGM 592_VALG

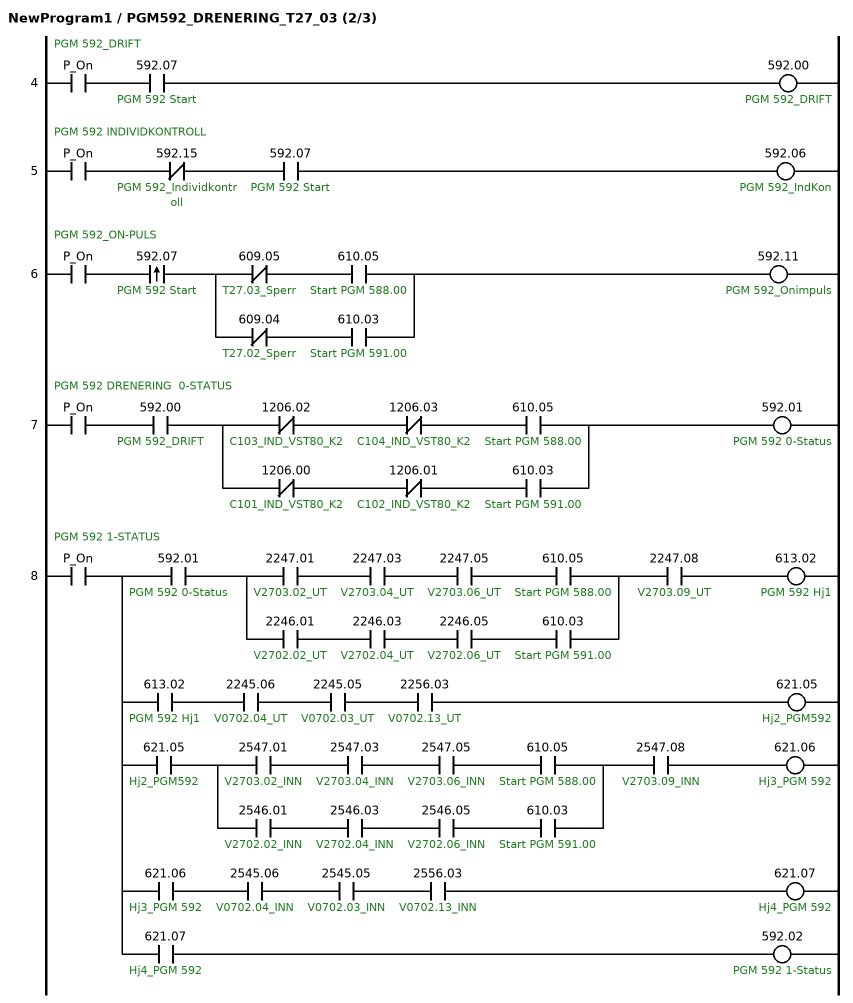
; rung 4: PGM 592_DRIFT
LD P_On
AND 592.07  ; PGM 592 Start
OUT 592.00  ; PGM 592_DRIFT
; rung 5: PGM 592 INDIVIDKONTROLL
LD P_On
ANDNOT 592.15  ; PGM 592_Individkontroll
AND 592.07  ; PGM 592 Start
OUT 592.06  ; PGM 592_IndKon
; rung 6: PGM 592_ON-PULS
LD P_On
@AND 592.07  ; PGM 592 Start
LDNOT 609.05  ; T27.03_Sperr
AND 610.05  ; Start PGM 588.00
LDNOT 609.04  ; T27.02_Sperr
AND 610.03  ; Start PGM 591.00
ORLD
ANDLD
OUT 592.11  ; PGM 592_Onimpuls
; rung 7: PGM 592 DRENERING  0-STATUS
LD P_On
AND 592.00  ; PGM 592_DRIFT
LDNOT 1206.02  ; C103_IND_VST80_K2
ANDNOT 1206.03  ; C104_IND_VST80_K2
AND 610.05  ; Start PGM 588.00
LDNOT 1206.00  ; C101_IND_VST80_K2
ANDNOT 1206.01  ; C102_IND_VST80_K2
AND 610.03  ; Start PGM 591.00
ORLD
ANDLD
OUT 592.01  ; PGM 592 0-Status
; rung 8: PGM 592 1-STATUS
LD P_On
OUT TR0
AND 592.01  ; PGM 592 0-Status
LD 2247.01  ; V2703.02_UT
AND 2247.03  ; V2703.04_UT
AND 2247.05  ; V2703.06_UT
AND 610.05  ; Start PGM 588.00
LD 2246.01  ; V2702.02_UT
AND 2246.03  ; V2702.04_UT
AND 2246.05  ; V2702.06_UT
AND 610.03  ; Start PGM 591.00
ORLD
ANDLD
AND 2247.08  ; V2703.09_UT
OUT 613.02  ; PGM 592 Hj1
LD TR0
AND 613.02  ; PGM 592 Hj1
AND 2245.06  ; V0702.04_UT
AND 2245.05  ; V0702.03_UT
AND 2256.03  ; V0702.13_UT
OUT 621.05  ; Hj2_PGM592
LD TR0
AND 621.05  ; Hj2_PGM592
LD 2547.01  ; V2703.02_INN
AND 2547.03  ; V2703.04_INN
AND 2547.05  ; V2703.06_INN
AND 610.05  ; Start PGM 588.00
LD 2546.01  ; V2702.02_INN
AND 2546.03  ; V2702.04_INN
AND 2546.05  ; V2702.06_INN
AND 610.03  ; Start PGM 591.00
ORLD
ANDLD
AND 2547.08  ; V2703.09_INN
OUT 621.06  ; Hj3_PGM 592
LD TR0
AND 621.06  ; Hj3_PGM 592
AND 2545.06  ; V0702.04_INN
AND 2545.05  ; V0702.03_INN
AND 2556.03  ; V0702.13_INN
OUT 621.07  ; Hj4_PGM 592
LD TR0
AND 621.07  ; Hj4_PGM 592
OUT 592.02  ; PGM 592 1-Status

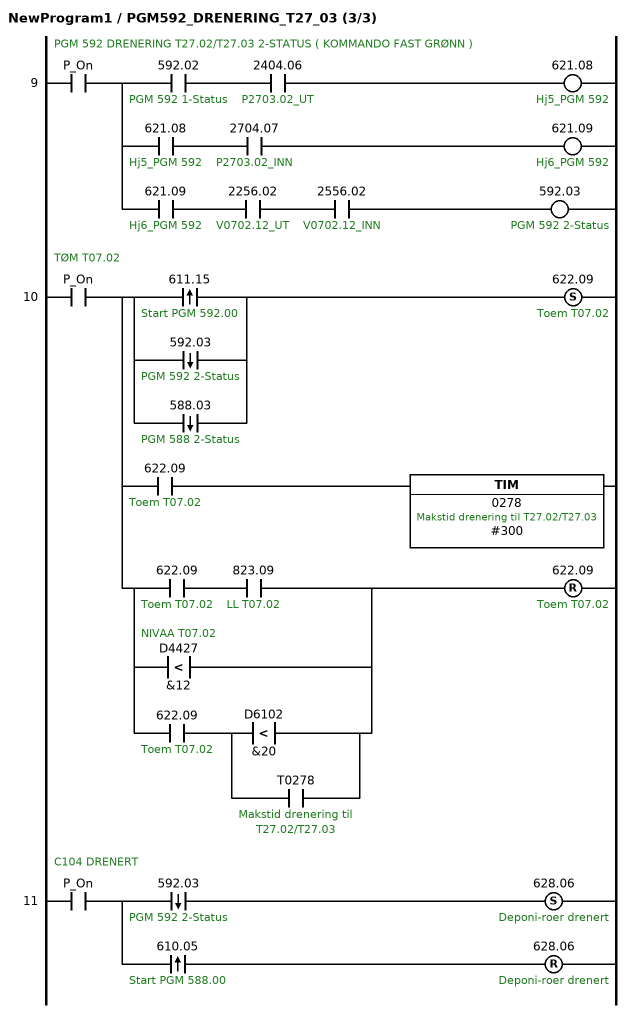
; rung 9: PGM 592 DRENERING T27.02/T27.03 2-STATUS ( KOMMANDO FAST GRØNN )
LD P_On
OUT TR0
AND 592.02  ; PGM 592 1-Status
AND 2404.06  ; P2703.02_UT
OUT 621.08  ; Hj5_PGM 592
LD TR0
AND 621.08  ; Hj5_PGM 592
AND 2704.07  ; P2703.02_INN
OUT 621.09  ; Hj6_PGM 592
LD TR0
AND 621.09  ; Hj6_PGM 592
AND 2256.02  ; V0702.12_UT
AND 2556.02  ; V0702.12_INN
OUT 592.03  ; PGM 592 2-Status
; rung 10: TØM T07.02
LD P_On
OUT TR0
@LD 611.15  ; Start PGM 592.00
%OR 592.03  ; PGM 592 2-Status
%OR 588.03  ; PGM 588 2-Status
ANDLD
SET 622.09  ; Toem T07.02
LD TR0
AND 622.09  ; Toem T07.02
TIM 0278 #300  ; Makstid drenering til T27.02/T27.03
LD TR0
LD 622.09  ; Toem T07.02
AND 823.09  ; LL T07.02
OR<(310) D4427 &12  ; NIVAA T07.02
LD 622.09  ; Toem T07.02
LD<(310) D6102 &20
OR T0278  ; Makstid drenering til T27.02/T27.03
ANDLD
ORLD
ANDLD
RSET 622.09  ; Toem T07.02
; rung 11: C104 DRENERT
LD P_On
OUT TR0
%AND 592.03  ; PGM 592 2-Status
SET 628.06  ; Deponi-roer drenert
LD TR0
@AND 610.05  ; Start PGM 588.00
RSET 628.06  ; Deponi-roer drenert

### Section PGM593_KONTAINER_T27_03

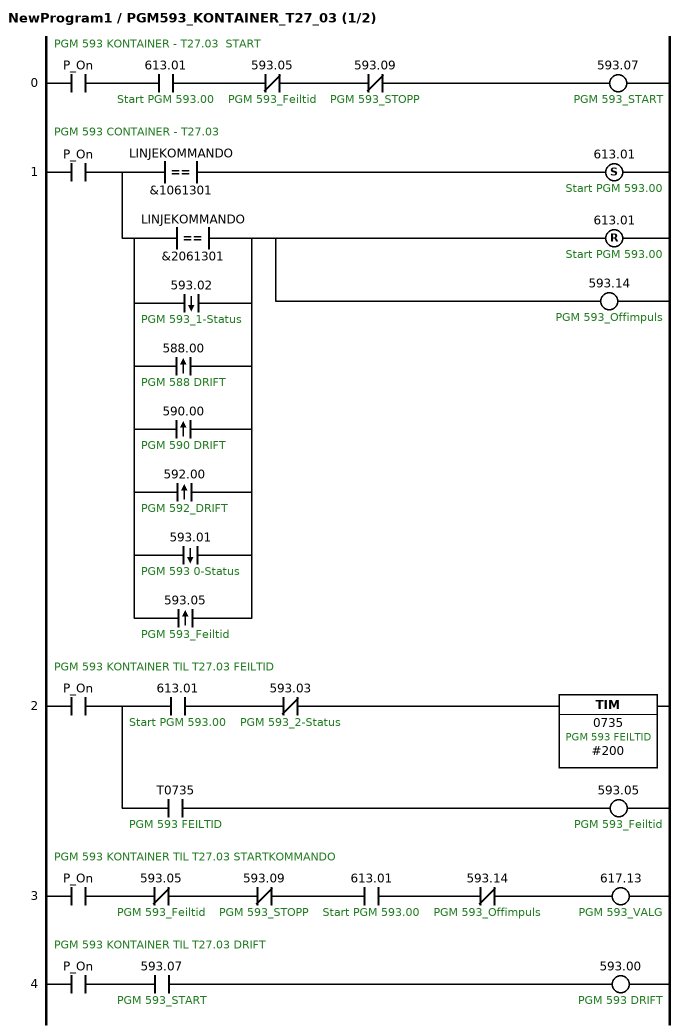
; rung 0: PGM 593 KONTAINER - T27.03  START
LD P_On
AND 613.01  ; Start PGM 593.00
ANDNOT 593.05  ; PGM 593_Feiltid
ANDNOT 593.09  ; PGM 593_STOPP
OUT 593.07  ; PGM 593_START
; rung 1: PGM 593 CONTAINER - T27.03
LD P_On
OUT TR0
AND=L(301) LINJEKOMMANDO &1061301
SET 613.01  ; Start PGM 593.00
LD TR0
LD=L(301) LINJEKOMMANDO &2061301
%OR 593.02  ; PGM 593_1-Status
@OR 588.00  ; PGM 588 DRIFT
@OR 590.00  ; PGM 590 DRIFT
@OR 592.00  ; PGM 592_DRIFT
%OR 593.01  ; PGM 593 0-Status
@OR 593.05  ; PGM 593_Feiltid
ANDLD
RSET 613.01  ; Start PGM 593.00
OUT 593.14  ; PGM 593_Offimpuls
; rung 2: PGM 593 KONTAINER TIL T27.03 FEILTID
LD P_On
OUT TR0
AND 613.01  ; Start PGM 593.00
ANDNOT 593.03  ; PGM 593_2-Status
TIM 0735 #200  ; PGM 593 FEILTID
LD TR0
AND T0735  ; PGM 593 FEILTID
OUT 593.05  ; PGM 593_Feiltid
; rung 3: PGM 593 KONTAINER TIL T27.03 STARTKOMMANDO
LD P_On
ANDNOT 593.05  ; PGM 593_Feiltid
ANDNOT 593.09  ; PGM 593_STOPP
AND 613.01  ; Start PGM 593.00
ANDNOT 593.14  ; PGM 593_Offimpuls
OUT 617.13  ; PGM 593_VALG
; rung 4: PGM 593 KONTAINER TIL T27.03 DRIFT
LD P_On
AND 593.07  ; PGM 593_START
OUT 593.00  ; PGM 593 DRIFT

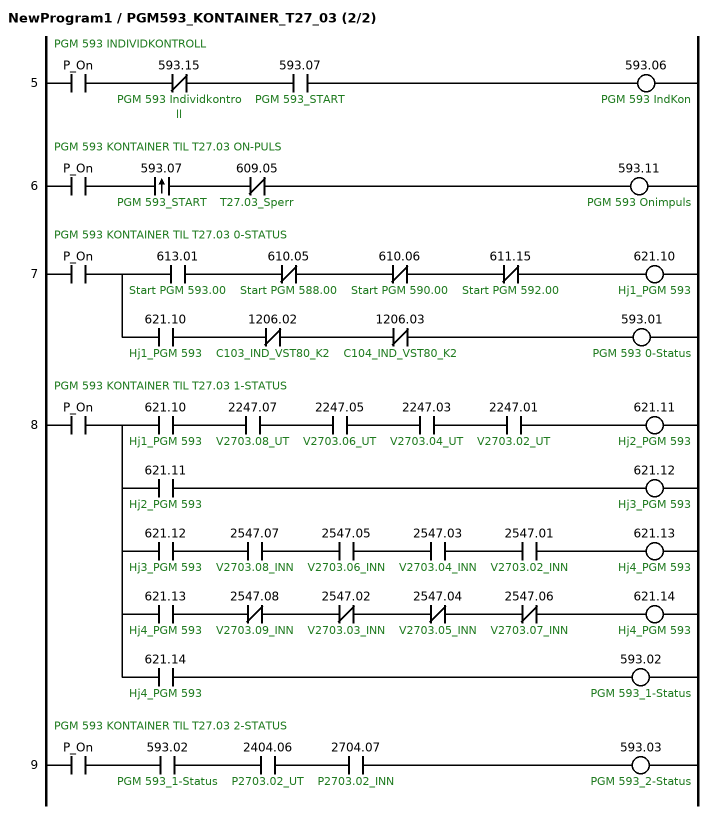
; rung 5: PGM 593 INDIVIDKONTROLL
LD P_On
ANDNOT 593.15  ; PGM 593 Individkontroll
AND 593.07  ; PGM 593_START
OUT 593.06  ; PGM 593 IndKon
; rung 6: PGM 593 KONTAINER TIL T27.03 ON-PULS
LD P_On
@AND 593.07  ; PGM 593_START
ANDNOT 609.05  ; T27.03_Sperr
OUT 593.11  ; PGM 593 Onimpuls
; rung 7: PGM 593 KONTAINER TIL T27.03 0-STATUS
LD P_On
OUT TR0
AND 613.01  ; Start PGM 593.00
ANDNOT 610.05  ; Start PGM 588.00
ANDNOT 610.06  ; Start PGM 590.00
ANDNOT 611.15  ; Start PGM 592.00
OUT 621.10  ; Hj1_PGM 593
LD TR0
AND 621.10  ; Hj1_PGM 593
ANDNOT 1206.02  ; C103_IND_VST80_K2
ANDNOT 1206.03  ; C104_IND_VST80_K2
OUT 593.01  ; PGM 593 0-Status
; rung 8: PGM 593 KONTAINER TIL T27.03 1-STATUS
LD P_On
OUT TR0
AND 621.10  ; Hj1_PGM 593
AND 2247.07  ; V2703.08_UT
AND 2247.05  ; V2703.06_UT
AND 2247.03  ; V2703.04_UT
AND 2247.01  ; V2703.02_UT
OUT 621.11  ; Hj2_PGM 593
LD TR0
AND 621.11  ; Hj2_PGM 593
OUT 621.12  ; Hj3_PGM 593
LD TR0
AND 621.12  ; Hj3_PGM 593
AND 2547.07  ; V2703.08_INN
AND 2547.05  ; V2703.06_INN
AND 2547.03  ; V2703.04_INN
AND 2547.01  ; V2703.02_INN
OUT 621.13  ; Hj4_PGM 593
LD TR0
AND 621.13  ; Hj4_PGM 593
ANDNOT 2547.08  ; V2703.09_INN
ANDNOT 2547.02  ; V2703.03_INN
ANDNOT 2547.04  ; V2703.05_INN
ANDNOT 2547.06  ; V2703.07_INN
OUT 621.14  ; Hj4_PGM 593
LD TR0
AND 621.14  ; Hj4_PGM 593
OUT 593.02  ; PGM 593_1-Status
; rung 9: PGM 593 KONTAINER TIL T27.03 2-STATUS
LD P_On
AND 593.02  ; PGM 593_1-Status
AND 2404.06  ; P2703.02_UT
AND 2704.07  ; P2703.02_INN
OUT 593.03  ; PGM 593_2-Status

### Section L1_L2_AUTODREN

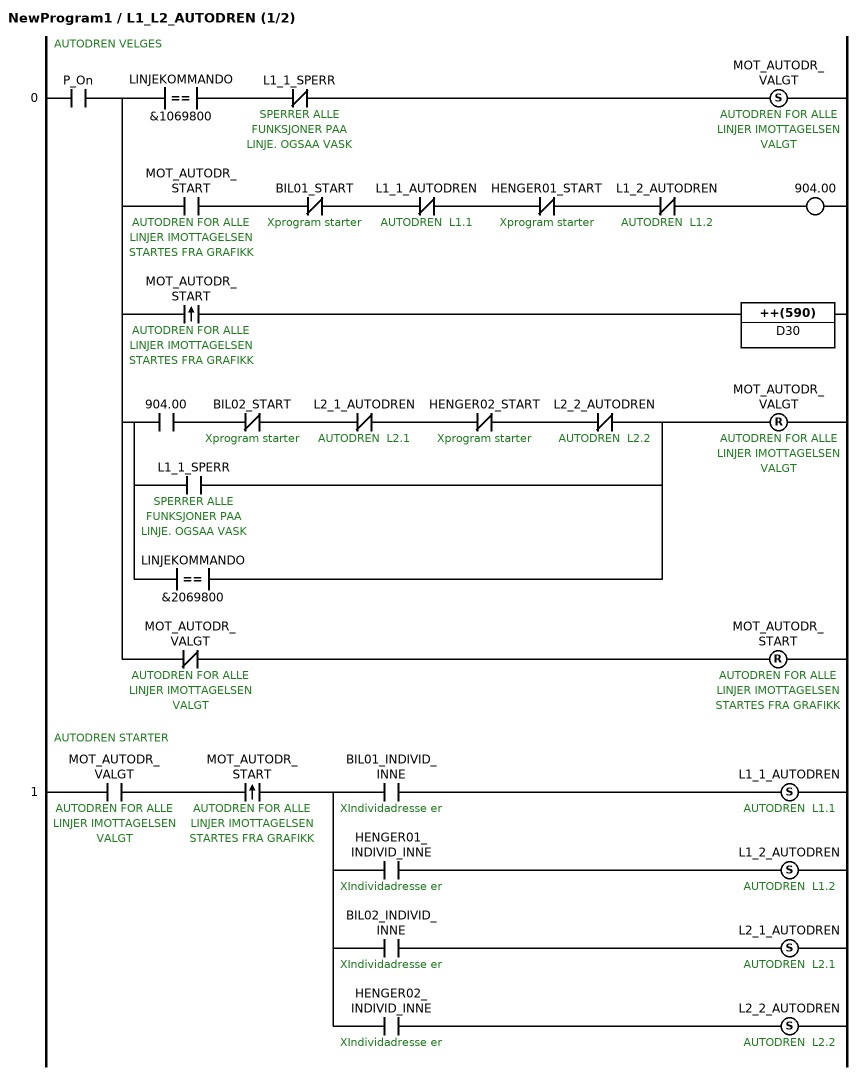
; rung 0: AUTODREN VELGES
LD P_On
OUT TR0
AND=L(301) LINJEKOMMANDO &1069800
ANDNOT L1_1_SPERR  ; SPERRER ALLE FUNKSJONER PAA LINJE. OGSAA VASK
SET MOT_AUTODR_VALGT  ; AUTODREN FOR ALLE LINJER IMOTTAGELSEN VALGT
LD TR0
AND MOT_AUTODR_START  ; AUTODREN FOR ALLE LINJER IMOTTAGELSEN STARTES FRA GRAFIKK
ANDNOT BIL01_START  ; Xprogram starter
ANDNOT L1_1_AUTODREN  ; AUTODREN  L1.1
ANDNOT HENGER01_START  ; Xprogram starter
ANDNOT L1_2_AUTODREN  ; AUTODREN  L1.2
OUT 904.00
LD TR0
@AND MOT_AUTODR_START  ; AUTODREN FOR ALLE LINJER IMOTTAGELSEN STARTES FRA GRAFIKK
++(590) D30
LD TR0
LD 904.00
ANDNOT BIL02_START  ; Xprogram starter
ANDNOT L2_1_AUTODREN  ; AUTODREN  L2.1
ANDNOT HENGER02_START  ; Xprogram starter
ANDNOT L2_2_AUTODREN  ; AUTODREN  L2.2
OR L1_1_SPERR  ; SPERRER ALLE FUNKSJONER PAA LINJE. OGSAA VASK
OR=L(301) LINJEKOMMANDO &2069800
ANDLD
RSET MOT_AUTODR_VALGT  ; AUTODREN FOR ALLE LINJER IMOTTAGELSEN VALGT
LD TR0
ANDNOT MOT_AUTODR_VALGT  ; AUTODREN FOR ALLE LINJER IMOTTAGELSEN VALGT
RSET MOT_AUTODR_START  ; AUTODREN FOR ALLE LINJER IMOTTAGELSEN STARTES FRA GRAFIKK
; rung 1: AUTODREN STARTER
LD MOT_AUTODR_VALGT  ; AUTODREN FOR ALLE LINJER IMOTTAGELSEN VALGT
@AND MOT_AUTODR_START  ; AUTODREN FOR ALLE LINJER IMOTTAGELSEN STARTES FRA GRAFIKK
OUT TR0
AND BIL01_INDIVID_INNE  ; XIndividadresse er
SET L1_1_AUTODREN  ; AUTODREN  L1.1
LD TR0
AND HENGER01_INDIVID_INNE  ; XIndividadresse er
SET L1_2_AUTODREN  ; AUTODREN  L1.2
LD TR0
AND BIL02_INDIVID_INNE  ; XIndividadresse er
SET L2_1_AUTODREN  ; AUTODREN  L2.1
LD TR0
AND HENGER02_INDIVID_INNE  ; XIndividadresse er
SET L2_2_AUTODREN  ; AUTODREN  L2.2

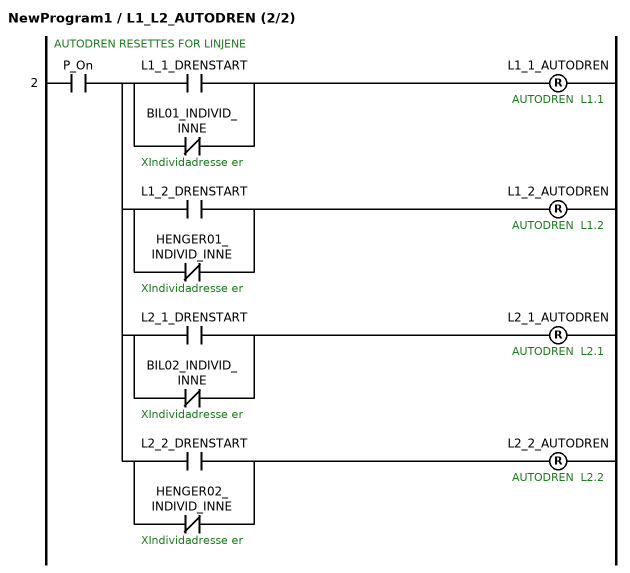
; rung 2: AUTODREN RESETTES FOR LINJENE
LD P_On
OUT TR0
LD L1_1_DRENSTART
ORNOT BIL01_INDIVID_INNE  ; XIndividadresse er
ANDLD
RSET L1_1_AUTODREN  ; AUTODREN  L1.1
LD TR0
LD L1_2_DRENSTART
ORNOT HENGER01_INDIVID_INNE  ; XIndividadresse er
ANDLD
RSET L1_2_AUTODREN  ; AUTODREN  L1.2
LD TR0
LD L2_1_DRENSTART
ORNOT BIL02_INDIVID_INNE  ; XIndividadresse er
ANDLD
RSET L2_1_AUTODREN  ; AUTODREN  L2.1
LD TR0
LD L2_2_DRENSTART
ORNOT HENGER02_INDIVID_INNE  ; XIndividadresse er
ANDLD
RSET L2_2_AUTODREN  ; AUTODREN  L2.2

### Section L1_1_STATUS

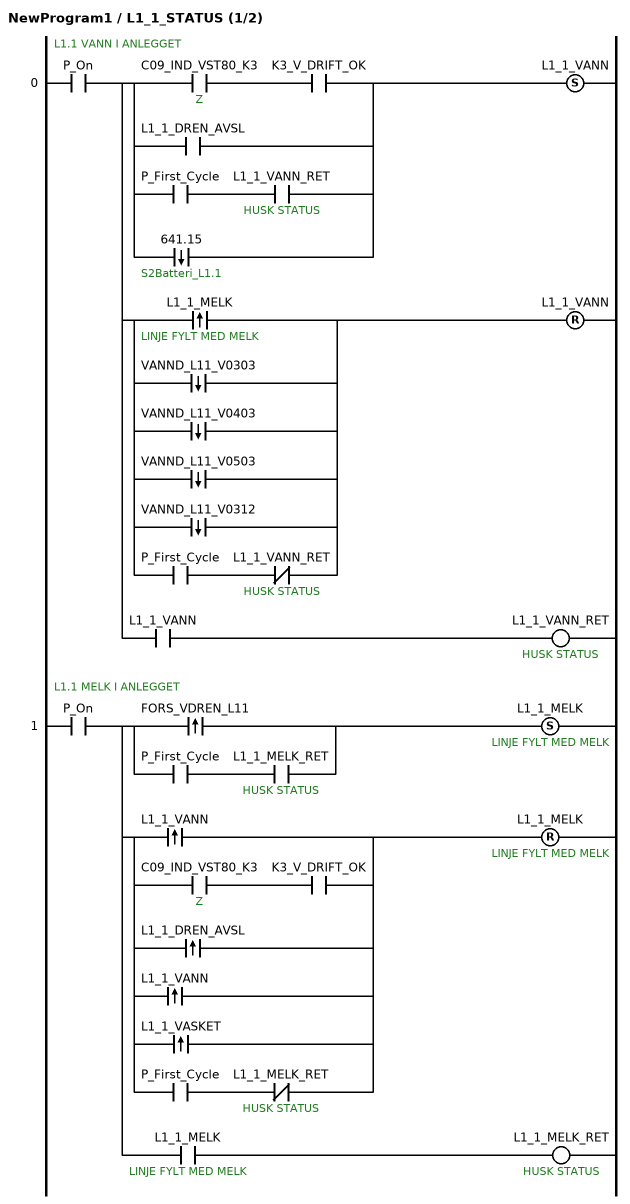
; rung 0: L1.1 VANN I ANLEGGET
LD P_On
OUT TR0
LD C09_IND_VST80_K3  ; Z
AND K3_V_DRIFT_OK
OR L1_1_DREN_AVSL
LD P_First_Cycle
AND L1_1_VANN_RET  ; HUSK STATUS
ORLD
%OR 641.15  ; S2Batteri_L1.1
ANDLD
SET L1_1_VANN
LD TR0
@LD L1_1_MELK  ; LINJE FYLT MED MELK
%OR VANND_L11_V0303
%OR VANND_L11_V0403
%OR VANND_L11_V0503
%OR VANND_L11_V0312
LD P_First_Cycle
ANDNOT L1_1_VANN_RET  ; HUSK STATUS
ORLD
ANDLD
RSET L1_1_VANN
LD TR0
AND L1_1_VANN
OUT L1_1_VANN_RET  ; HUSK STATUS
; rung 1: L1.1 MELK I ANLEGGET
LD P_On
OUT TR0
@LD FORS_VDREN_L11
LD P_First_Cycle
AND L1_1_MELK_RET  ; HUSK STATUS
ORLD
ANDLD
SET L1_1_MELK  ; LINJE FYLT MED MELK
LD TR0
@LD L1_1_VANN
LD C09_IND_VST80_K3  ; Z
AND K3_V_DRIFT_OK
ORLD
@OR L1_1_DREN_AVSL
@OR L1_1_VANN
@OR L1_1_VASKET
LD P_First_Cycle
ANDNOT L1_1_MELK_RET  ; HUSK STATUS
ORLD
ANDLD
RSET L1_1_MELK  ; LINJE FYLT MED MELK
LD TR0
AND L1_1_MELK  ; LINJE FYLT MED MELK
OUT L1_1_MELK_RET  ; HUSK STATUS

